PROGRAM P_TaskHandling
VAR
	// Robot task status informaiton
	// UR3
	fbUR3TaskStatusInfo : FB_mbReadRobotTaskStatusInfo := (Robot := 'UR3');
	stUR3TaskStatus : ST_RobotTaskStatusInfo;
	// UR5
	fbUR5TaskStatusInfo : FB_mbReadRobotTaskStatusInfo := (Robot := 'UR5');
	stUR5TaskStatus : ST_RobotTaskStatusInfo;
	
	// Task Triggers
	StopAssignment_ftrig : F_TRIG;
	// UR3
	UR3TaskActive_rtrig : R_TRIG; // Task assigned (including positioning movements)
	UR3TaskComplete_ftrig : F_TRIG; // Task reported complete
	UR3ActionStart_rtrig : R_TRIG; // robot positioning for task over, part interaction begins
	UR3ActionComplete_ftrig : F_TRIG; // part interaction ends
	//UR5
	UR5TaskActive_rtrig : R_TRIG; // Task assigned (including positioning movements)
	UR5TaskComplete_ftrig : F_TRIG; // Task reported complete
	UR5ActionStart_rtrig : R_TRIG; // robot positioning for task over, part interaction begins
	UR5ActionComplete_ftrig : F_TRIG; // part interaction ends
	
	// General use indexes and counters
	nMaxTimeInWF : REAL;
	nWorkFixtureIndex : INT;
	nInputFixtureIndex : INT;
	nOutputFixtureIndex : INT;
	
	// UR3 Task State Macine
	eUR3TaskState : E_RobotTaskStates;
	
	// UR3 Active Task Targets
	nUR3TargetWorkFixtureIndex : INT;
	nUR3TargetWorkframe : WORD;
	nUR3TargetTask : WORD;
	nUR3TargetPart : WORD;
	
	// UR5 Task State Macine
	eUR5TaskState : E_RobotTaskStates;
	
	// UR5 Active Task Targets
	nUR5TargetWorkFixtureIndex : INT;
	nUR5TargetInputFixtureIndex : INT;
	nUR5TargetOutputFixtureIndex : INT;
	nUR5TargetPickFrame : WORD;
	nUR5TargetPlaceFrame : WORD;
	nUR5TargetTask: WORD; // 1 for input 2 for output
	sUR5TargetTask: STRING;
	nUR5TargetPart : WORD;
	
	// Task writing functionblocks
	fbWriteUR3Task : FB_mbWriteRobotTask := (Robot := 'UR3');
	fbWriteUR5Task : FB_mbWriteRobotTask := (Robot := 'UR5');
	fbUR3Resume : FB_mbWriteSingleReg := (Robot := 'UR3', Register := 145, Value := 1);
	fbUR5Resume : FB_mbWriteSingleReg := (Robot := 'UR5', Register := 145, Value := 1);
	
	// Position Check variables
	bPosCheckNext : BOOL;
	nTaskType: INT := 1;
	bPosCheckAssignedUR3: BOOL;
	bPosCheckAssignedUR5: BOOL;
	bPosCheckCompleteUR3: BOOL;
	bPosCheckCompleteUR5: BOOL;
	nUR3PosCheckIndex : UINT := 1;
	nUR5PosCheckIndex : UINT := 1;
	
	bTestWait: BOOL;
END_VAR

(* =======================================================
Update veriables on every cycle
Multiple states are calculated on each cycle to aid in task assignment and tracking
======================================================= *)
// Update Task Status Information
fbUR3TaskStatusInfo(stTaskStatusInfo => stUR3TaskStatus);
fbUR5TaskStatusInfo(stTaskStatusInfo => stUR5TaskStatus);

// Triggers and Event Tracking
// Position Check Triggers
	IF Global.bEnablePosCheck THEN
		IF Global.bForcePosCheck OR Global.nPartsSincePosCheck >= Global.nPosCheckThreshold THEN
			bPosCheckNext := TRUE;
		END_IF
	END_IF
	// Reset Pos Check founter if it has been assigned for both robots
	IF bPosCheckCompleteUR3 AND bPosCheckCompleteUR5 THEN
		// if required trigger post check processing here
		Global.nPartsSincePosCheck := 0;
		bPosCheckAssignedUR3 := FALSE;
		bPosCheckAssignedUR5 := FALSE;
		bPosCheckCompleteUR3 := FALSE;
		bPosCheckCompleteUR5 := FALSE;
		bPosCheckNext := FALSE;
		Global.bForcePosCheck := FALSE;
	END_IF
// Stop Process Triggers
	StopAssignment_ftrig(CLK := Global.bActivateTaskAssignment);
	// Global interrupt
	// Interrupts
	IF StopAssignment_ftrig.Q THEN
		IF eUR3TaskState = E_RobotTaskStates.TaskSelection OR eUR3TaskState = E_RobotTaskStates.TaskTypeSelection THEN
			eUR3TaskState := E_RobotTaskStates.Idle;
		END_IF
		IF eUR5TaskState = E_RobotTaskStates.TaskSelection OR eUR5TaskState = E_RobotTaskStates.TaskTypeSelection THEN
			eUR5TaskState := E_RobotTaskStates.Idle;
		END_IF
	END_IF
//UR3 Task Triggers
	// Watch for UR3 task to be assigned
	UR3TaskActive_rtrig(CLK := stUR3TaskStatus.bInTask);
	// Watch for UR3 task to complete
	UR3TaskComplete_ftrig(CLK := stUR3TaskStatus.bInTask);
	// Watch for UR3 to start task action
	UR3ActionStart_rtrig(CLK := stUR3TaskStatus.bPerformingTaskAction);
	// Watch for UR3 to complete task action
	UR3ActionComplete_ftrig(CLK := stUR3TaskStatus.bPerformingTaskAction);
//UR5 Task Triggers
	// Watch for UR3 task to be assigned
	UR5TaskActive_rtrig(CLK := stUR5TaskStatus.bInTask);
	// Watch for UR3 task to complete
	UR5TaskComplete_ftrig(CLK := stUR5TaskStatus.bInTask);
	// Watch for UR3 to start task action
	UR5ActionStart_rtrig(CLK := stUR5TaskStatus.bPerformingTaskAction);
	// Watch for UR3 to complete task action
	UR5ActionComplete_ftrig(CLK := stUR5TaskStatus.bPerformingTaskAction);

// Calcualte part Time in Fixture
// Cycle through every workfixture
FOR nWorkFixtureIndex := 1 TO Global.nNumWorkFixtures DO
	// Calculate part times on every loop
	IF Global.arrWorkFixtures[nWorkFixtureIndex].stPart.bExists THEN
		Global.arrWorkFixtures[nWorkFixtureIndex].stPart.ntTimeInWorkfixture := 
			(Global.nCurrentTime - Global.arrWorkFixtures[nWorkFixtureIndex].stPart.ntInputPartPlaced)/10000000;
	ELSE
		Global.arrWorkFixtures[nWorkFixtureIndex].stPart.ntTimeInWorkfixture := 0;
	END_IF
END_FOR

// Update task type strings for visualization
IF eUR5TaskState = E_RobotTaskStates.TaskExecution THEN
	IF nUR5TargetTask = 1 THEN
		sUR5TargetTask := 'Input';
	ELSIF nUR5TargetTask = 2 THEN
		sUR5TargetTask := 'Output';
	END_IF
ELSE
	sUR5TargetTask := 'N/A';
END_IF


(* =======================================================
A state machine is used to handle the task state of the UR3 robot.
	Possible states include:
		- Idle - wait until process is in a mode to execute tasks
		- Task Type Selection - this is used to select between a drawing task or a measurement task. More can be added in the future
		- Task Selection - if no task is being executed, assesing if a task should be assigned
		- Task Assignment - packaging a task and transmititng it to the robot
		- Task Assignment Wait - waiting for task to be written to robot
		- Task Execution - waiting for robot to complete assigned task before going back to Idle
======================================================= *)
CASE eUR3TaskState OF
	E_RobotTaskStates.Idle: // Decides what to do based on system mode
		IF Global.bActivateTaskAssignment AND Global_Safety.UR3RedIND THEN
			eUR3TaskState := E_RobotTaskStates.TaskTypeSelection;
		END_IF
		// Reset Targets
		nUR3TargetWorkFixtureIndex := 0;
		nUR3TargetWorkframe := 0;
		nUR3TargetTask := 0;
		Global.bUR3InTask := FALSE;
	E_RobotTaskStates.TaskTypeSelection: // Should a position check test be performed
		IF bPosCheckNext AND NOT Global.bUR5InTask THEN
			IF NOT Global.bPosSensorReserved AND NOT bPosCheckCompleteUR3 THEN
				// Set Task Variables 
				nUR3TargetTask := 0; // 0 for Pos Check Program on robots
				Global.bPosSensorReserved := TRUE;
				bPosCheckAssignedUR3 := TRUE;
				nUR3PosCheckIndex := 1; // Index Value for Assignment of Sensor Inputs - Reset to 1
				eUR3TaskState := E_RobotTaskStates.TaskAssignment;
			END_IF
		ELSIF NOT bPosCheckNext THEN // else check if a different task that can be assigned
			// If a part exists and is not complete move to task selection
			IF Global.arrWorkFixtures[1].stPart.bExists AND NOT Global.arrWorkFixtures[1].stPart.bComplete THEN // If WF1 has a part that is not complete
				eUR3TaskState := E_RobotTaskStates.TaskSelection;
			ELSIF  Global.arrWorkFixtures[2].stPart.bExists AND NOT Global.arrWorkFixtures[2].stPart.bComplete THEN
				eUR3TaskState := E_RobotTaskStates.TaskSelection;
			END_IF
		END_IF
	E_RobotTaskStates.TaskSelection: // Monitoring and deciding if a task should be assigned
		// Reset MaxPartLagTime to help find longest lag time
		nMaxTimeInWF := 0;
		// Reset Targets
		nUR3TargetWorkFixtureIndex := 0;
		nUR3TargetWorkframe := 0;
		nUR3TargetTask := 0;
		// For each possible active workfixture
		FOR nWorkFixtureIndex := 1 TO Global.nNumWorkFixtures DO
			// If statement to identify if fixture/part can be worked on
			IF 	Global.arrWorkFixtures[nWorkFixtureIndex].stPart.bExists // part exists
			AND	NOT Global.arrWorkFixtures[nWorkFixtureIndex].stPart.bComplete // part not complete
			AND	NOT Global.arrWorkFixtures[nWorkFixtureIndex].bReserved THEN // fixture not reserved
				// Check to see if identified eligable part has been waiting the longest
				IF Global.arrWorkFixtures[nWorkFixtureIndex].stPart.ntTimeInWorkfixture > nMaxTimeInWF THEN
					// update max part lag time
					nMaxTimeInWF := Global.arrWorkFixtures[nWorkFixtureIndex].stPart.ntTimeInWorkfixture;
					// Record task, workframe and workfixture index
					nUR3TargetWorkframe := Global.arrWorkFixtures[nWorkFixtureIndex].nWorkframe;
					nUR3TargetPart := Global.arrWorkFixtures[nWorkFixtureIndex].stPart.nPartNumber;
					nUR3TargetWorkFixtureIndex := nWorkFixtureIndex;
					// if a viable target is found assign task
					eUR3TaskState := E_RobotTaskStates.TaskAssignment;
				END_IF
			END_IF
		END_FOR
		
		// Choose Task number 
		nUR3TargetTask := Global.nActiveUR3Task + 1; // 1 added for array indexing on radio button visu (starts at 0)
		(*
		FOR FUTURE VERSIONS - IF TASK IS TIED TO PART TYPE 
		Part type is stored in the following locaiton:
		Global.arrWorkFixtures[nUR3TargetWorkFixtureIndex].stPart.nPartType;
		*)
		
	E_RobotTaskStates.TaskAssignment: // Transmitting task to robot
		Global.bUR3InTask := TRUE;
		(* This section has two parts. 1) PLC handling and part tracking and 2) handling assignment to robot. *)
		// PLC Handling
		Global.arrWorkFixtures[nUR3TargetWorkFixtureIndex].bReserved := TRUE;
		
		// Robot Assignment Setup Handling
		fbWriteUR3Task.Task := nUR3TargetTask;
		fbWriteUR3Task.Workframe1 := nUR3TargetWorkframe;
		fbWriteUR3Task.PartNumber := nUR3TargetPart;
		fbWriteUR3Task.bExecute := TRUE;
		
		// Advance to waiting for assignment completion
		eUR3TaskState := E_RobotTaskStates.TaskAssignment_Wait;
	
	E_RobotTaskStates.TaskAssignment_Wait: 	// Waiting for task to be written
		IF NOT fbWriteUR3Task.bBusy THEN
			fbWriteUR3Task.bExecute :=FALSE;
			// record task assignment
			Global.arrWorkFixtures[nUR3TargetWorkFixtureIndex].stPart.ntTaskAssigned := Global.nCurrentTime;
			// change states
			eUR3TaskState := E_RobotTaskStates.TaskExecution;
		END_IF
			
	E_RobotTaskStates.TaskExecution: // Monitoring for completion of task
		// Recording Time at events
		IF UR3ActionStart_rtrig.Q THEN
			IF nUR3TargetTask = 0 THEN
				// record IO state here
				Global.UR3PosCheck[nUR3PosCheckIndex] := Global.bPosSensorState;
				nUR3PosCheckIndex := nUR3PosCheckIndex + 1;
				// tell robot to resume task
				fbUR3Resume.bExecute := TRUE;
			ELSE
				Global.arrWorkFixtures[nUR3TargetWorkFixtureIndex].stPart.ntTaskActionStart := Global.nCurrentTime;
			END_IF
		END_IF
		
		IF UR3ActionComplete_ftrig.Q THEN
			IF nUR3TargetTask = 0 THEN
				; // do noting
			ELSE
				Global.arrWorkFixtures[nUR3TargetWorkFixtureIndex].stPart.ntTaskActionComplete := Global.nCurrentTime;
			END_IF
		END_IF
		
		IF UR3TaskComplete_ftrig.Q THEN
			IF nUR3TargetTask = 0 THEN // If task completed was a pos check
				bPosCheckCompleteUR3 := TRUE;
				Global.bPosSensorReserved := FALSE;
				// (FOR UR integrated sensor) Global.UR3PosCheck := F_Word_To_16Bool(stUR3TaskStatus.nPosCheckValue);
			ELSE
				Global.arrWorkFixtures[nUR3TargetWorkFixtureIndex].stPart.bComplete := TRUE;
				Global.arrWorkFixtures[nUR3TargetWorkFixtureIndex].bReserved := FALSE;
				// Record Complete
				Global.arrWorkFixtures[nUR3TargetWorkFixtureIndex].stPart.ntTaskComplete := Global.nCurrentTime;
			END_IF
			// Go back to idle state
			eUR3TaskState := E_RobotTaskStates.Idle;
		END_IF
END_CASE

(* =======================================================
UR5
A state machine is used to handle the task state of the UR5 robot.
	Possible states include:
		- Idle - wait until process is in a mode to execute tasks
		- Task Selection - if no task is being executed, assesing if a task should be assigned
		- Task Assignment - packaging a task and transmititng it to the robot
		- Task Assignment Wait - waiting for task to be written to robot
		- Task Execution - waiting for robot to complete assigned task before going back to Idle
======================================================= *)
CASE eUR5TaskState OF
	E_RobotTaskStates.Idle: // Decides what to do based on system mode
		IF Global.bActivateTaskAssignment AND Global_Safety.UR5RedIND THEN
			eUR5TaskState := E_RobotTaskStates.TaskTypeSelection;
		END_IF
		// Reset Targets
		nUR5TargetWorkFixtureIndex := 0;
		nUR5TargetInputFixtureIndex := 0;
		nUR5TargetOutputFixtureIndex := 0;
		nUR5TargetPickFrame := 0;
		nUR5TargetPlaceFrame := 0;
		nUR5TargetTask := 0;
		nMaxTimeInWF := 0;
		Global.bUR5InTask := FALSE;
	E_RobotTaskStates.TaskTypeSelection: // Should a position check test be performed
		IF bPosCheckNext AND NOT Global.bUR3InTask THEN
			// Choose Task number 
			IF NOT Global.bPosSensorReserved AND NOT bPosCheckCompleteUR5 THEN
				nUR5TargetTask := 0; // 0 for Pos Check Program on robots
				Global.bPosSensorReserved := TRUE;
				bPosCheckAssignedUR5 := TRUE;
				nUR5PosCheckIndex := 1; // Index Value for Assignment of Sensor Inputs - Reset to 1
				eUR5TaskState := E_RobotTaskStates.TaskAssignment;
			END_IF
		ELSIF NOT bPosCheckNext THEN  
			// else it is a different task that must be assigned
			// If an input part exists or a complete part exists
			IF Global.arrInputFixtures[1].stPart.bExists OR Global.arrWorkFixtures[1].stPart.bComplete OR Global.arrWorkFixtures[2].stPart.bComplete THEN 
				eUR5TaskState := E_RobotTaskStates.TaskSelection;
			END_IF
		END_IF
	E_RobotTaskStates.TaskSelection: // Monitoring and deciding if a task should be assigned
		// OUTPUT - Find possible part OUTPUTS
		nUR5TargetPickFrame := 0;
		nUR5TargetPlaceFrame := 0;
		// For each possible active workfixture
		FOR nWorkFixtureIndex := 1 TO Global.nNumWorkFixtures DO
			IF Global.arrWorkFixtures[nWorkFixtureIndex].stPart.bExists // part exists
			AND Global.arrWorkFixtures[nWorkFixtureIndex].stPart.bComplete // part is complete (ready for output)
			AND NOT Global.arrWorkFixtures[nWorkFixtureIndex].bReserved THEN // fixture is not reserved
				// Determine if it has been waiting the longest (FIFO)
				IF Global.arrWorkFixtures[nWorkFixtureIndex].stPart.ntTimeInWorkfixture > nMaxTimeInWF THEN
					// update max part lag time
					nMaxTimeInWF := Global.arrWorkFixtures[nWorkFixtureIndex].stPart.ntTimeInWorkfixture;
					// Record task, workframe and workfixture index
					nUR5TargetWorkFixtureIndex := nWorkFixtureIndex;
					nUR5TargetPart := Global.arrWorkFixtures[nWorkFixtureIndex].stPart.nPartNumber;
					nUR5TargetPickFrame := Global.arrWorkFixtures[nWorkFixtureIndex].nWorkframe;
				END_IF
			END_IF
		END_FOR
		// For each possible output fixture
		FOR nOutputFixtureIndex := 1 TO Global.nNumOutputFixtures DO
			// find first available input part (in order, NO FIFO)
			IF NOT Global.arrOutputFixtures[nOutputFixtureIndex].stPart.bExists THEN
				// Record target information
				nUR5TargetOutputFixtureIndex := nOutputFixtureIndex;
				nUR5TargetPlaceFrame := Global.arrOutputFixtures[nOutputFixtureIndex].nWorkframe;
				// if a viable target is found assign task
			END_IF
			IF nUR5TargetPlaceFrame > 0 THEN
					// exit for loop
					EXIT;
			END_IF
		END_FOR
		// assign task type if a task was found
		IF nUR5TargetPickFrame <> 0 AND nUR5TargetPlaceFrame <> 0 THEN // pick and place found
			nUR5TargetTask := 2; // 2 for output task
			eUR5TaskState := E_RobotTaskStates.TaskAssignment;
		END_IF
		// INPUT - If output is not assigned find possible INPUTS
		
		IF nUR5TargetTask <> 2 THEN
			nUR5TargetPickFrame := 0;
			nUR5TargetPlaceFrame := 0;
			// check if each work fixture is empty
			FOR nWorkFixtureIndex := 1 TO Global.nNumWorkFixtures DO
				IF NOT Global.arrWorkFixtures[nWorkFixtureIndex].stPart.bExists // no part in fixture
				AND NOT Global.arrWorkFixtures[nWorkFixtureIndex].bReserved THEN // fixture is not reserved
					// record target informaiton
					nUR5TargetWorkFixtureIndex := nWorkFixtureIndex;
					nUR5TargetPlaceFrame := Global.arrWorkFixtures[nWorkFixtureIndex].nWorkframe;
				END_IF
				IF nUR5TargetPlaceFrame > 0 THEN
					// exit for loop
					EXIT;
				END_IF
			END_FOR
			// check for available part in input
			FOR nInputFixtureIndex := 1 TO Global.nNumInputFixtures DO
				// find first available input part (in order, NO FIFO)
				IF 	Global.arrInputFixtures[nInputFixtureIndex].stPart.bExists THEN
					// Record target information
					nUR5TargetInputFixtureIndex := nInputFixtureIndex;
					nUR5TargetPart := Global.arrInputFixtures[nInputFixtureIndex].stPart.nPartNumber;
					nUR5TargetPickFrame := Global.arrInputFixtures[nInputFixtureIndex].nWorkframe;
				END_IF
				IF nUR5TargetPickFrame > 0 THEN
					// exit for loop
					EXIT;
				END_IF
			END_FOR
			// check if task was assigned
			IF nUR5TargetPickFrame <> 0 AND nUR5TargetPlaceFrame <> 0 THEN
				nUR5TargetTask := 1; // 1 for input task
				eUR5TaskState := E_RobotTaskStates.TaskAssignment;
			END_IF
		END_IF
	E_RobotTaskStates.TaskAssignment: // Transmitting task to robot
		(* This section has two parts. 1) handling PLC tracking side and 2) handling assignment to robot. *)
		// PLC Handling
		Global.bUR5InTask  := TRUE;
		IF nUR5TargetTask = 1 THEN // If input task
			Global.arrInputFixtures[nUR5TargetInputFixtureIndex].bReserved := TRUE;
			// Record task information
			Global.arrInputFixtures[nUR5TargetInputFixtureIndex].stPart.nInputPosition := nUR5TargetPickFrame;
			Global.arrInputFixtures[nUR5TargetInputFixtureIndex].stPart.nWorkFixture := nUR5TargetPlaceFrame;
		ELSIF nUR5TargetTask = 2 THEN // If output task
			Global.arrOutputFixtures[nUR5TargetOutputFixtureIndex].bReserved := TRUE;
			// Record task information
			Global.arrWorkFixtures[nUR5TargetWorkFixtureIndex].stPart.nOutputPosition := nUR5TargetPlaceFrame;
		END_IF
		
		Global.arrWorkFixtures[nUR5TargetWorkFixtureIndex].bReserved := TRUE;
		
		
		// Robot Assignment Setup Handling
		fbWriteUR5Task.Task := nUR5TargetTask;
		fbWriteUR5Task.Workframe1 := nUR5TargetPickFrame;
		fbWriteUR5Task.Workframe2 := nUR5TargetPlaceFrame;
		fbWriteUR5Task.PartNumber := nUR5TargetPart;
		fbWriteUR5Task.bExecute := TRUE;
		
		// Advance to waiting for assignment completion
		eUR5TaskState := E_RobotTaskStates.TaskAssignment_Wait;
	
	E_RobotTaskStates.TaskAssignment_Wait: 	// Waiting for task to be written
		IF NOT fbWriteUR5Task.bBusy THEN
			fbWriteUR5Task.bExecute :=FALSE;
			// record assignment time
			IF nUR5TargetTask = 1 THEN // If input task
				Global.arrInputFixtures[nUR5TargetInputFixtureIndex].stPart.ntPickFromInputAssigned := Global.nCurrentTime;
			ELSIF nUR5TargetTask = 2 THEN // If output task
				Global.arrWorkFixtures[nUR5TargetWorkFixtureIndex].stPart.ntPickFromWFAssigned := Global.nCurrentTime;
			END_IF
			
			// change states
			eUR5TaskState := E_RobotTaskStates.TaskExecution;
		END_IF
			
	E_RobotTaskStates.TaskExecution: // Monitoring for completion of task
		// Handle task events
		IF UR5ActionStart_rtrig.Q THEN // when action starts
			IF nUR5TargetTask = 0 THEN
				// record IO state here
				Global.UR5PosCheck[nUR5PosCheckIndex] := Global.bPosSensorState;
				nUR5PosCheckIndex := nUR5PosCheckIndex + 1;
				// tell robot to resume task
				fbUR5Resume.bExecute := TRUE;
			// record Action start time and handle part movement
			ELSIF nUR5TargetTask = 1 THEN // If input task
				Global.arrInputFixtures[nUR5TargetInputFixtureIndex].stPart.ntInputPartPicked := Global.nCurrentTime;
				Global.stPartInTransit := Global.arrInputFixtures[nUR5TargetInputFixtureIndex].stPart;
				Global.arrInputFixtures[nUR5TargetInputFixtureIndex].stPart := Global.stNullPart;
			ELSIF nUR5TargetTask = 2 THEN // If output task
				Global.arrWorkFixtures[nUR5TargetWorkFixtureIndex].stPart.ntOutputPartPicked := Global.nCurrentTime;
				Global.stPartInTransit := Global.arrWorkFixtures[nUR5TargetWorkFixtureIndex].stPart;
				Global.arrWorkFixtures[nUR5TargetWorkFixtureIndex].stPart := Global.stNullPart;
			END_IF
		END_IF
		IF UR5ActionComplete_ftrig.Q THEN
			IF nUR5TargetTask = 0 THEN
				; // do noting
			// record Action Complete time and handle part movement
			ELSIF nUR5TargetTask = 1 THEN // If input task
				Global.arrWorkFixtures[nUR5TargetWorkFixtureIndex].stPart := Global.stPartInTransit;
				Global.arrWorkFixtures[nUR5TargetWorkFixtureIndex].stPart.ntInputPartPlaced := Global.nCurrentTime;
				Global.stPartInTransit := Global.stNullPart;
			ELSIF nUR5TargetTask = 2 THEN // If output task
				Global.arrOutputFixtures[nUR5TargetOutputFixtureIndex].stPart := Global.stPartInTransit;
				Global.arrOutputFixtures[nUR5TargetOutputFixtureIndex].stPart.ntOutputPartPlaced := Global.nCurrentTime;
				Global.stPartInTransit := Global.stNullPart;
			END_IF
		END_IF
		
		IF UR5TaskComplete_ftrig.Q THEN
			// record Action Complete time and handle part movement
			IF nUR5TargetTask = 0 THEN // If task completed was a pos check
				bPosCheckCompleteUR5 := TRUE;
				Global.bPosSensorReserved := FALSE;
				// Global.UR5PosCheck := F_Word_To_16Bool(stUR5TaskStatus.nPosCheckValue);
			ELSIF nUR5TargetTask = 1 THEN // If input task
				Global.arrWorkFixtures[nUR5TargetWorkFixtureIndex].stPart.ntPlaceInWFComplete := Global.nCurrentTime;
				Global.arrWorkFixtures[nUR5TargetWorkFixtureIndex].bReserved := FALSE;
				Global.arrInputFixtures[nUR5TargetInputFixtureIndex].bReserved := FALSE;
			ELSIF nUR5TargetTask = 2 THEN // If output task
				Global.arrOutputFixtures[nUR5TargetOutputFixtureIndex].stPart.ntPlaceInOutputComplete := Global.nCurrentTime;
				Global.arrOutputFixtures[nUR5TargetOutputFixtureIndex].bReserved := FALSE;
				Global.arrWorkFixtures[nUR5TargetWorkFixtureIndex].bReserved := FALSE;
				// Pos Check Part Counting
				Global.nPartsSincePosCheck := Global.nPartsSincePosCheck + 1;
			END_IF
			// Go back to idle state
			eUR5TaskState := E_RobotTaskStates.Idle;
		END_IF
END_CASE

(* =======================================================
Function block Calls
======================================================= *)
fbWriteUR3Task();
fbWriteUR5Task();
fbUR3Resume();
fbUR5Resume();

END_PROGRAM

(* stored: Version 1.1.0.1, ProductVersion 3.1.4020.12
   POU P_TaskHandling: Id {7d4036fb-bc78-45ef-ba00-c501dee2fa25}, SpecialFunc None *)
